INTERFACE I_ForwardEnumerator EXTENDS I_Disposable

PROPERTY PUBLIC IsValid : BOOL
GET
END_GET
END_PROPERTY

METHOD PUBLIC MoveNext : BOOL
VAR_INPUT
END_VAR
END_METHOD

METHOD PUBLIC TryGet : BOOL;
VAR_INPUT
	Destination : ANY;
END_VAR
END_METHOD

METHOD PUBLIC TryGetTo : BOOL;
VAR_INPUT
	Destination : PVOID;
	DestinationSize : UDINT;
END_VAR
END_METHOD

END_INTERFACE

(* stored: Version 1.1.0.1, ProductVersion 3.1.4024.12
   Itf I_ForwardEnumerator: Id {e9757b38-1996-45e6-a6c8-96fd1404a343}
   Property IsValid: Id {ca3b8f11-a3d3-4a38-972a-a72264c1ee16}
   Get Get: Id {a6419129-5d78-4c7b-92a5-0b3480f2ac1b}
   Method MoveNext: Id {9260f718-b451-4949-bbf4-855569ebd9d6}
   Method TryGet: Id {5edda5f9-87aa-4554-95ac-2b6a71d4c829}
   Method TryGetTo: Id {0dcbd2bc-5561-4b8e-8861-f42207a07a4a} *)
